// TIA Portal V17 export
// export: Created 2024-09-02T12:50:40.16223Z, ExportSetting WithDefaults, DisplayName Totally Integrated Automation Portal, DisplayVersion V17, DisplayName TIA Portal Openness, DisplayVersion V17, DisplayName TIA Portal Version Control Interface, DisplayVersion V17, DisplayName STEP 7 Professional, DisplayVersion V17, DisplayName STEP 7 Safety, DisplayVersion V17, DisplayName WinCC Professional, DisplayVersion V17
TYPE "Scania_typ_Results"
// stored: IsFailsafeCompliant false
   STRUCT
      WorkFinishedTimeStamp : Date_And_Time;
      StatusOpeation : Array[1..16] of "Scania_typ_Status";
   END_STRUCT;
END_TYPE
